FUNCTION_BLOCK DualOut_2_DO (* Service Interface Function Block Type *)
  (* Function: All Outputs; Description: this maps to QX *)
  (* Version 1.0, 2018-12-05, Jose Cabral *)
  (* Version 1.1, 2022-08-04, Franz Höpfinger, HR Agrartechnik GmbH *)
  (* Version 1.2, 2023-01-05, Franz Höpfinger, HR Agrartechnik GmbH *)
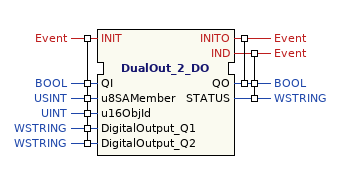
  EVENT_INPUT
    INIT WITH QI, u8SAMember, u16ObjId, DigitalOutput_Q1, DigitalOutput_Q2; (* Service Initialization *)
  END_EVENT
  EVENT_OUTPUT
    INITO WITH QO; (* Initialization Confirm *)
    IND WITH QO, STATUS; (* Indication from Resource *)
  END_EVENT
  VAR_INPUT
    QI : BOOL; (* Event Input Qualifier *)
    u8SAMember : USINT := 255; (* Dummy !, set to 255 if in doubt. 0 deactivates FB. *)
    u16ObjId : UINT := 65535; (* Dummy ! set to 65535 if in Doubt. 0 deactivates FB. *)
    DigitalOutput_Q1 : WSTRING := "DigitalOutput_Q1";
    DigitalOutput_Q2 : WSTRING := "DigitalOutput_Q2";
  END_VAR
  VAR_OUTPUT
    QO : BOOL; (* Event Output Qualifier *)
    STATUS : WSTRING; (* Service Status *)
  END_VAR
END_FUNCTION_BLOCK
